TYPE "PLCtoMES_ProcessingExchange"
VERSION : 0.1
   STRUCT
      "P-ProcessingPartID" : String[48];
      "P-ProcessingReq" : Bool;
      Reserve : Array[1..248] of Byte;
   END_STRUCT;

END_TYPE

